FUNCTION_BLOCK Skill_LoadDeliverReturn EXTENDS FB_Skill
VAR_INPUT
	Rob: POINTER TO FB_ROB_AMR;
	sPickReference: STRING;
END_VAR
VAR_OUTPUT
	
END_VAR
VAR
	
	ActiveBAFinished: BOOL;
END_VAR

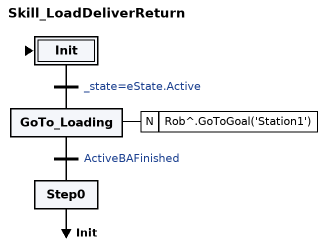
INITIAL_STEP Init:
END_STEP
TRANSITION FROM Init TO GoTo_Loading
    := _state=eState.Active;
END_TRANSITION
STEP GoTo_Loading:
    Rob^.GoToGoal('Station1')(N);
END_STEP
TRANSITION FROM GoTo_Loading TO Step0
    := ActiveBAFinished;
END_TRANSITION
STEP Step0:
END_STEP
// no transition between Step0 and Init

END_FUNCTION_BLOCK

(* stored: Version 1.1.0.1, ProductVersion 3.1.4026.18
   POU Skill_LoadDeliverReturn: Id {8977347b-02ee-433d-9081-1576e654bc94}, SpecialFunc None *)
